TYPE sBogie :
STRUCT
	
	A : sWX_Side;
	B : sWX_Side;
	
	//Vert	: ClearpathPosition;
	//Rot		: ClearpathPosition;
	//Clamp	: ClearpathPOsition;
	bFileCheckOk 	: BOOL;
	CurrentJob 		: MoldJob;
	
	bArmsAtTravelPos 	: BOOL;
	
	bEnabled : BOOL;
	
	//Conveyor Signals
	ConveyorLoadPos : BOOL;

END_STRUCT
END_TYPE

(* stored: Version 1.1.0.1, ProductVersion 3.1.4024.12
   DUT sBogie: Id {6e2cd502-5e05-41e8-bb2a-3ec617a1fb96} *)
